{attribute 'GeneratedUsingTerminal: EJ1918-0000-0017'}
{attribute addProperty BoxType "EJ1918-0000-0017"}
{attribute addProperty Id "FSOEAT %Q*FSOE_878484619"}
{attribute addProperty CRC "3778608309"}
{attribute addProperty Size "9"}
TYPE FSoE_Outputs_E138FCB5 EXTENDS OutputBase_10CEE7DE :
STRUCT
	{attribute addProperty Name "FSOE"}
	FSOE AT %Q* : FSOE_87848461;
END_STRUCT
END_TYPE

(* stored: Version 1.2.0.0, ProductVersion 3.1.4024.9
   DUT FSoE_Outputs_E138FCB5: Id {ab594199-c935-42f1-8c93-196a7bc63760} *)
